// TIA Portal V19 export
TYPE "LEXCHANGETRAY_typeLogistics_toRollerDeliver"
// stored: Access Published
   STRUCT
      feedback : "LEXCHANGETRAY_typeLogistics_toRollerFeedback";   // 允许物流线排料
      req : "LEXCHANGETRAY_typeLogistics_toRollerReq";
   END_STRUCT;
END_TYPE
